Staubli VAL3: RobotStatus.dtx

public JointSpace jointSpace
  [0]
    JointPos jointPos
      [0]
        jointRx jp
    JointVel jointVel
      [0]
        num jv[6]
    JointAccel jointAccel
      [0]
        num ja[6]
    JointForce jointForce
      [0]
        num jf[6]
public CartesianSpace cartesianSpace
  [0]
    CartesianPos cartesianPos
      [0]
        pointRx cp
    CartesianVel cartesianVel
      [0]
        num resVel
        num cv[6]
    CartesianAccel cartesianAccel
      [0]
        num ca[6]
        num resAccel
    CartesianForce cartesianForce
      [0]
        num cf[6]
        num resForce
